// TIA Portal V20 export
VAR_GLOBAL   // PLC tag table "Default tag table_2"
END_VAR
